FUNCTION_BLOCK FB_CommandChangeSuspend EXTENDS FB_CommandChange IMPLEMENTS ITF_CommandChange
VAR

END_VAR

(*			
	EVERDE sp. z o.o.
	Rafał Osajda		03.11.2025		TC 4024.66
	Test czy można zmienić stan lub tryb i zwraca czy można i uruchamia zmianę
*)
METHOD PUBLIC Execute : BOOL
VAR_INPUT
	iNumberOfCommand	: INT;
END_VAR
IF (THIS^.itfSaMController.GetState () = E_BaseMachineState.Execute) THEN		// sprawdzenie czy jesteśmy w dobrym stanie dla tego rozkazu
	IF (THIS^.itfSaMController.IsStateInModeEnabled (eNewState := E_BaseMachineState.Suspending)) THEN	//test czy stan do którego chcemy przejśc jest właczony dla tego trybu
		THIS^.itfSaMController.ChangeStateTo (eNewState := E_BaseMachineState.Suspending);
	ELSE
		THIS^.EventSetActive (iNumber := 5);	//stan docelowy jest wylaczony w tym trybie
	END_IF
ELSE
	THIS^.EventSetActive (iNumber := 4);	//ten rozkaz nie obsluguje tego stanu
END_IF
END_METHOD

METHOD FB_init : BOOL
VAR_INPUT
	bInitRetains : BOOL; // if TRUE, the retain variables are initialized (warm start / cold start)
	bInCopyCode : BOOL;  // if TRUE, the instance afterwards gets moved into the copy code (online change)
END_VAR
THIS^.SetText (eLocation := E_BaseLocation.pl, wsDescription := "Command change state - Suspend");
THIS^.SetText (eLocation := E_BaseLocation.en, wsDescription := "Command change state - Suspend");
THIS^.SetText (eLocation := E_BaseLocation.de, wsDescription := "Command change state - Suspend");
THIS^.SetName (stName := THIS^.GetTexts ());
END_METHOD

END_FUNCTION_BLOCK

(* stored: Version 1.1.0.1
   POU FB_CommandChangeSuspend: Id {48484d22-ae57-0719-2adb-4a264957724b}, SpecialFunc None
   Method Execute: Id {802cbb7f-9193-0075-2d6e-1fb41b0e3655}
   Method FB_init: Id {b5801e7d-e0c6-0514-120e-ac73f18d720c} *)
